(* PLC project CounterTest *)
(* stored: creationDateTime 2024-01-01T00:00:00, modificationDateTime 2024-01-01T00:00:00 *)

PROGRAM Main
  VAR
    X001 : BOOL;
    X002 : BOOL;
    X003 : BOOL;
    Y001 : BOOL;
    Y002 : BOOL;
    CTU1 : CTU;
    CTD1 : CTD;
  END_VAR

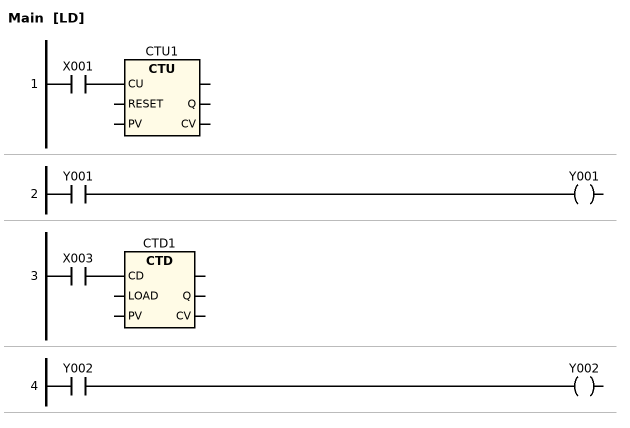
(* LD diagram, written out as Structured Text *)
Y001 := Y001;
Y002 := Y002;
CTU1(CU := X001);
CTD1(CD := X003);
END_PROGRAM

CONFIGURATION Config
  RESOURCE Res ON PLC
    TASK Main(INTERVAL := T#20ms, PRIORITY := 0);
    PROGRAM Main WITH Main : Main;
  END_RESOURCE
END_CONFIGURATION
